TYPE stPF_POINT :
STRUCT
	active_power: REAL;
	frequency: REAL;
END_STRUCT
END_TYPE

(* stored: Version 1.1.0.1, ProductVersion 3.1.4026.11
   DUT stPF_POINT: Id {5f392e7b-1477-4d3d-9be6-2630b6262df2} *)
